FUNCTION_BLOCK Test_StringSplitter_Splits_On_Tab EXTENDS TUnitTestBase
VAR
    StringSplitter : TStringSplitter;
END_VAR

Test_Started();

StringSplitter.Init(
    Str    := 'Bob$TCharles$TDavid',
    Delim1 := '$T',
    Delim2 := '');

Assertion.AssertEquals_STRING(
    Expected := 'Bob',
    Actual   := StringSplitter.GetNext(),
    ObjectName := _TestName,
    VariableName  := 'StringSplitter.GetNext()');

Assertion.AssertEquals_STRING(
    Expected := 'Charles',
    Actual   := StringSplitter.GetNext(),
    ObjectName := _TestName,
    VariableName  := 'StringSplitter.GetNext()');

Assertion.AssertEquals_STRING(
    Expected := 'David',
    Actual   := StringSplitter.GetNext(),
    ObjectName := _TestName,
    VariableName  := 'StringSplitter.GetNext()');


Test_Finished();

END_FUNCTION_BLOCK

(* stored: Version 1.1.0.1, ProductVersion 3.1.4024.3
   POU Test_StringSplitter_Splits_On_Tab: Id {86e3e891-db36-057f-3764-d41869894fb8}, SpecialFunc None *)
